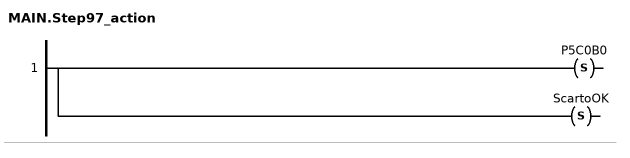
[picture p72: MAIN.Step97_action (LD)]
_LD_ (* Ladder Diagram *)
NETWORK 1
	* --- (S P5C0B0) (S ScartoOK)
_END_LD_
(* the same logic as Structured Text *)
(* Network 1 *)
P5C0B0 := TRUE;
ScartoOK := TRUE;
END_ACTION

ACTION ResetScarto_action:
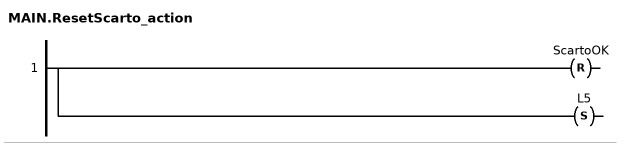
_LD_ (* Ladder Diagram *)
NETWORK 1
	* --- (R ScartoOK) (S L5)
_END_LD_
(* the same logic as Structured Text *)
(* Network 1 *)
ScartoOK := FALSE;
L5 := TRUE;
END_ACTION

ACTION ScartaPezzo_action:
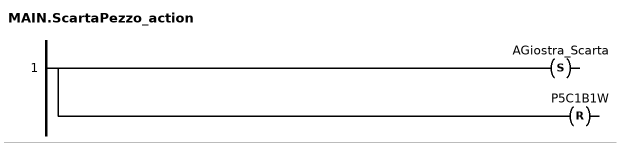
_LD_ (* Ladder Diagram *)
NETWORK 1
	* --- (S AGiostra_Scarta) (R P5C1B1W)
_END_LD_
(* the same logic as Structured Text *)
(* Network 1 *)
AGiostra_Scarta := TRUE;
P5C1B1W := FALSE;
END_ACTION

ACTION ugjvhavshva_action:
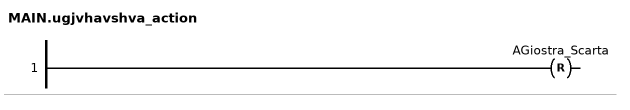
_LD_ (* Ladder Diagram *)
NETWORK 1
	* --- (R AGiostra_Scarta)
_END_LD_
(* the same logic as Structured Text *)
(* Network 1 *)
AGiostra_Scarta := FALSE;
END_ACTION

ACTION ResetL5_action:
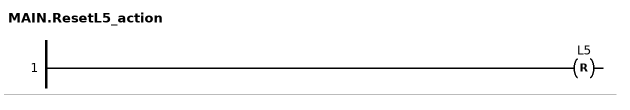
_LD_ (* Ladder Diagram *)
NETWORK 1
	* --- (R L5)
_END_LD_
(* the same logic as Structured Text *)
(* Network 1 *)
L5 := FALSE;
END_ACTION

ACTION Mantieni_action:
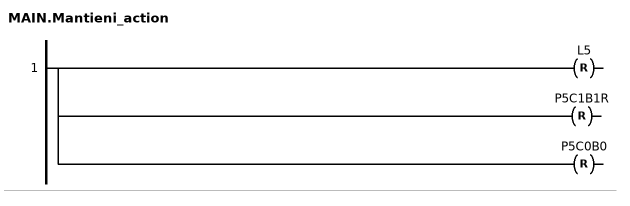
_LD_ (* Ladder Diagram *)
NETWORK 1
	* --- (R L5) (R P5C1B1R) (R P5C0B0)
_END_LD_
(* the same logic as Structured Text *)
(* Network 1 *)
L5 := FALSE;
P5C1B1R := FALSE;
P5C0B0 := FALSE;
END_ACTION

ACTION Rot13_action:
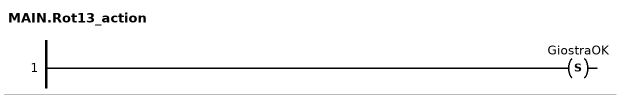
_LD_ (* Ladder Diagram *)
NETWORK 1
	* --- (S GiostraOK)
_END_LD_
(* the same logic as Structured Text *)
(* Network 1 *)
GiostraOK := TRUE;
END_ACTION

ACTION Step94_action:
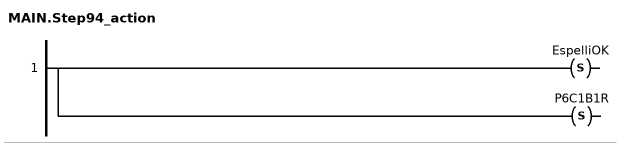
_LD_ (* Ladder Diagram *)
NETWORK 1
	* --- (S EspelliOK) (S P6C1B1R)
_END_LD_
(* the same logic as Structured Text *)
(* Network 1 *)
EspelliOK := TRUE;
P6C1B1R := TRUE;
END_ACTION

ACTION FermaSx_action:
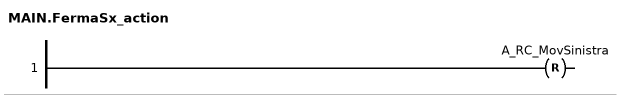
_LD_ (* Ladder Diagram *)
NETWORK 1
	* --- (R A_RC_MovSinistra)
_END_LD_
(* the same logic as Structured Text *)
(* Network 1 *)
A_RC_MovSinistra := FALSE;
END_ACTION

ACTION FermaDx_action:
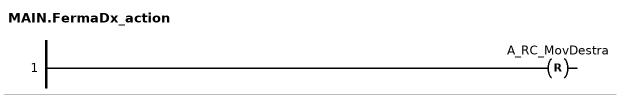
_LD_ (* Ladder Diagram *)
NETWORK 1
	* --- (R A_RC_MovDestra)
_END_LD_
(* the same logic as Structured Text *)
(* Network 1 *)
A_RC_MovDestra := FALSE;
END_ACTION

ACTION FermaDown_action:
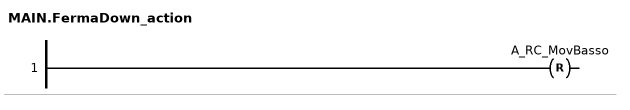
_LD_ (* Ladder Diagram *)
NETWORK 1
	* --- (R A_RC_MovBasso)
_END_LD_
(* the same logic as Structured Text *)
(* Network 1 *)
A_RC_MovBasso := FALSE;
END_ACTION

ACTION ContatoreRC_action:
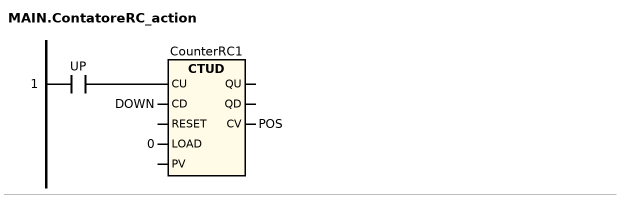
_LD_ (* Ladder Diagram *)
NETWORK 1
	[UP] - CounterRC1:CTUD(CU: *, CD: DOWN, RESET: , LOAD: 0, PV: , CV => POS)
_END_LD_
END_ACTION

ACTION ConversioneRC_action:
IF A_RC_MovDestra=TRUE
THEN UP :=S_RC_Encoder;
ELSIF A_RC_MovSinistra=TRUE
THEN DOWN :=S_RC_Encoder;
END_IF;

Z:=POS;
Z1:=WORD_TO_STRING(Z);
Z2:=CONCAT('16#',Z1);
Z3:=STRING_TO_INT(Z2);

IF Z3>16#0468 THEN
Bilancia:=TRUE;
ELSE Bilancia:=FALSE;
END_IF;

IF Z3<16#0393 THEN
Scivolo3:=TRUE;
ELSE Scivolo3:=FALSE;
END_IF;

IF Z3<16#0351 THEN
Scivolo2:=TRUE;
ELSE Scivolo2:=FALSE;
END_IF;

IF Z3<16#0315 THEN
Scivolo1:=TRUE;
ELSE Scivolo1:=FALSE;
END_IF;

IF Z3<16#0010 THEN
Partenza:=TRUE;
ELSE Partenza:=FALSE;
END_IF;
END_ACTION

ACTION ConvEst_action:
X1:=S_RC_Estensimetro;
X2:=WORD_TO_STRING(X1);
X3:=CONCAT('16#',X2);
IST:=STRING_TO_INT(X3);
IF IST>16#15470
THEN AltScivolo:=TRUE;
ELSE AltScivolo:=FALSE;
END_IF;
IF IST>16#24850
THEN AltFinale:=TRUE;
ELSE AltFinale:=FALSE;
END_IF;
IF IST<16#11300
THEN AltBase:=TRUE;
ELSE AltBase:=FALSE;
END_IF;
IF IST<16#10800
THEN AltBilancia:=TRUE;
ELSE AltBilancia:=FALSE;
END_IF;
END_ACTION

ACTION ResStart_action:
Start:=TRUE;
IF IST<16#25000 THEN
A_RC_MovAlto:=TRUE;
ELSE
A_RC_MovBasso:=TRUE;
END_IF;
END_ACTION

ACTION Ack2_action:
IF A_RC_MovAlto=TRUE THEN
  StopSali:=TRUE;
END_IF;

IF A_RC_MovBasso=TRUE THEN
  StopScendi:=TRUE;
END_IF;
END_ACTION

ACTION LivelloA_action:
IF IST>16#24800 THEN
   A_RC_MovAlto:=FALSE;
END_IF;
END_ACTION

ACTION LivelloB_action:
IF IST<16#25400 THEN
   A_RC_MovBasso:=FALSE;
END_IF;
END_ACTION

ACTION AvvioRSD_action:
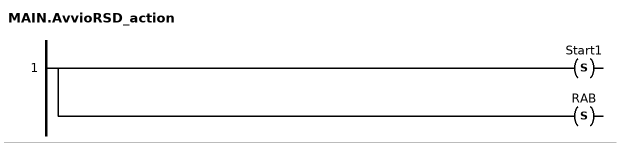
_LD_ (* Ladder Diagram *)
NETWORK 1
	* --- (S Start1) (S RAB)
_END_LD_
(* the same logic as Structured Text *)
(* Network 1 *)
Start1 := TRUE;
RAB := TRUE;
END_ACTION

ACTION ResStart1_action:
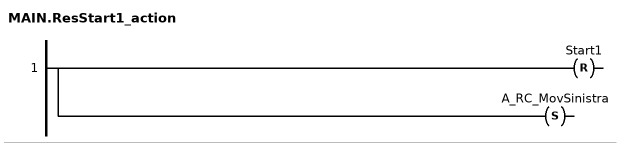
_LD_ (* Ladder Diagram *)
NETWORK 1
	* --- (R Start1) (S A_RC_MovSinistra)
_END_LD_
(* the same logic as Structured Text *)
(* Network 1 *)
Start1 := FALSE;
A_RC_MovSinistra := TRUE;
END_ACTION

ACTION Bounce_action:
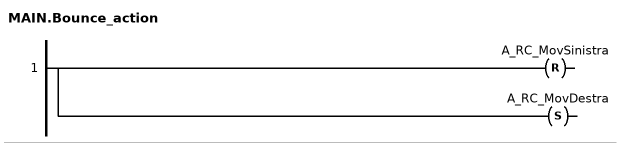
_LD_ (* Ladder Diagram *)
NETWORK 1
	* --- (R A_RC_MovSinistra) (S A_RC_MovDestra)
_END_LD_
(* the same logic as Structured Text *)
(* Network 1 *)
A_RC_MovSinistra := FALSE;
A_RC_MovDestra := TRUE;
END_ACTION

ACTION LivelloD_action:
IF Z3>16#005 THEN
A_RC_MovDestra:=FALSE;
END_IF;
END_ACTION

ACTION SetRSD_action:
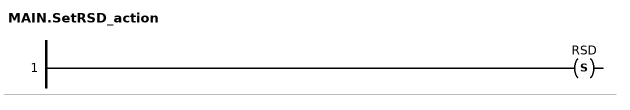
_LD_ (* Ladder Diagram *)
NETWORK 1
	* --- (S RSD)
_END_LD_
(* the same logic as Structured Text *)
(* Network 1 *)
RSD := TRUE;
END_ACTION

ACTION Step164_action:
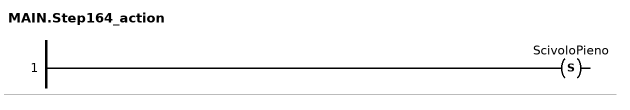
_LD_ (* Ladder Diagram *)
NETWORK 1
	* --- (S ScivoloPieno)
_END_LD_
(* the same logic as Structured Text *)
(* Network 1 *)
ScivoloPieno := TRUE;
END_ACTION

ACTION Step165_action:
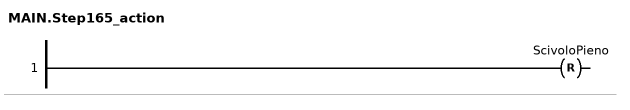
_LD_ (* Ladder Diagram *)
NETWORK 1
	* --- (R ScivoloPieno)
_END_LD_
(* the same logic as Structured Text *)
(* Network 1 *)
ScivoloPieno := FALSE;
END_ACTION

ACTION MovDVarC_action:
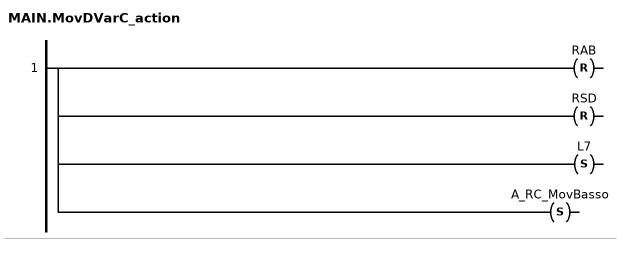
_LD_ (* Ladder Diagram *)
NETWORK 1
	* --- (R RAB) (R RSD) (S L7) (S A_RC_MovBasso)
_END_LD_
(* the same logic as Structured Text *)
(* Network 1 *)
RAB := FALSE;
RSD := FALSE;
L7 := TRUE;
A_RC_MovBasso := TRUE;
END_ACTION

ACTION StopBase_action:
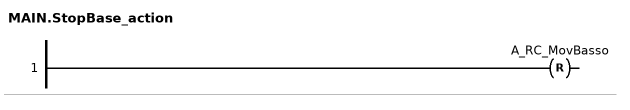
_LD_ (* Ladder Diagram *)
NETWORK 1
	* --- (R A_RC_MovBasso)
_END_LD_
(* the same logic as Structured Text *)
(* Network 1 *)
A_RC_MovBasso := FALSE;
END_ACTION

ACTION PinzaSet1_action:
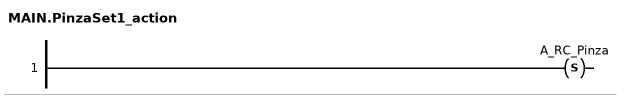
_LD_ (* Ladder Diagram *)
NETWORK 1
	* --- (S A_RC_Pinza)
_END_LD_
(* the same logic as Structured Text *)
(* Network 1 *)
A_RC_Pinza := TRUE;
END_ACTION

ACTION MovA_action:
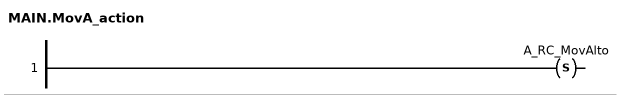
_LD_ (* Ladder Diagram *)
NETWORK 1
	* --- (S A_RC_MovAlto)
_END_LD_
(* the same logic as Structured Text *)
(* Network 1 *)
A_RC_MovAlto := TRUE;
END_ACTION

ACTION MovDRMovA_action:
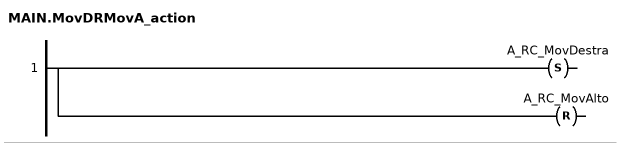
_LD_ (* Ladder Diagram *)
NETWORK 1
	* --- (S A_RC_MovDestra) (R A_RC_MovAlto)
_END_LD_
(* the same logic as Structured Text *)
(* Network 1 *)
A_RC_MovDestra := TRUE;
A_RC_MovAlto := FALSE;
END_ACTION

ACTION MovBRMovD_action:
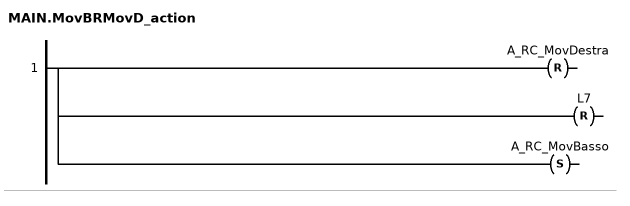
_LD_ (* Ladder Diagram *)
NETWORK 1
	* --- (R A_RC_MovDestra) (R L7) (S A_RC_MovBasso)
_END_LD_
(* the same logic as Structured Text *)
(* Network 1 *)
A_RC_MovDestra := FALSE;
L7 := FALSE;
A_RC_MovBasso := TRUE;
END_ACTION

ACTION LasciaPezzo_action:
